FUNCTION_BLOCK itfDetectImplement IMPLEMENTS itfDetect
VAR_INPUT
END_VAR
VAR_OUTPUT
END_VAR
VAR
	DetectSignal : BOOL;
END_VAR

{warning 'add property implementation'}
PROPERTY pDetectSignal : BOOL
GET
pDetectSignal := DetectSignal;
END_GET
SET
DetectSignal := pDetectSignal;
END_SET
END_PROPERTY

END_FUNCTION_BLOCK

(* stored: Version 1.1.0.1, ProductVersion 3.1.4024.12
   POU itfDetectImplement: Id {188124eb-46d1-43ca-a6ab-cdd97081cc06}, SpecialFunc None
   Property pDetectSignal: Id {b8b58071-26a9-4759-a020-388c05ae4184}
   Get Get: Id {a517cb68-b173-4cb0-b937-6d0a8a9b325b}
   Set Set: Id {81d31114-a1cd-464b-b8da-a948783a30ab} *)
